// TIA Portal V18 export
VAR_GLOBAL   // PLC tag table "Default tag table"
   ESTOP_Button AT %I0.0 : Bool;   // Emergency button
   JOGNEG_BTN_Z1 AT %I0.2 : Bool;   // Z1 - Jogging Negative -> In order to execute this, real button sholud be pressed
   JOGPOS_BTN_Z1 AT %I0.1 : Bool;   // Z1 - Jogging Positive -> In order to execute this, real button sholud be pressed
   JOGNEG_BTN_Z2 AT %I0.4 : Bool;   // Z2 - Jogging Negative -> In order to execute this, real button sholud be pressed
   JOGPOS_BTN_Z2 AT %I0.3 : Bool;   // Z2 - Jogging Positive -> In order to execute this, real button sholud be pressed
   SENSOR_DOOR AT %I0.5 : Bool;   // Door Sensor Front
   Load_Cell_Ink AT %IW66 : UInt;
   Load_Cell_Waste AT %IW64 : UInt;
   SENSOR_DOOR_2 AT %I0.6 : Bool;   // Door Sensor Front
   UV_Error_Signal AT %I0.7 : Bool;   // Error signal from UV lamp, 0-4 V error, 16-24 V ok;
   SENSOR_DOOR_3 AT %I1.0 : Bool;   // Door Sensor Side
   SENSOR_DOOR_4 AT %I1.1 : Bool;   // Door Sensor Side
   SENSOR_DOOR_5 AT %I1.2 : Bool;   // Door Sensor Fluid Supply
   SENSOR_DOOR_6 AT %I1.3 : Bool;   // Door Sensor Fluid Supply
   TemperatureSensor AT %IW116 : UInt;
   CappingSensor AT %IW118 : UInt;
   AnalogInput3 AT %IW120 : UInt;
   AnalogInput4 AT %IW122 : UInt;
   "Roller Encoder" AT %ID1000 : DWord;
   "STO-B_Output" AT %Q0.0 : Bool;   // Safty Torque Off , for CMMO [Port X3, Pin ..]and CMMP in order to release a break
   Roller_Output AT %Q0.6 : Bool;
   Heater_Output AT %Q1.0 : Bool;   // Heater: ON/OFF_PLC/3.2B; %Q1.0
   LED_1_Output AT %Q0.4 : Bool;
   LED_2_Output AT %Q0.5 : Bool;
   Heater_PWM_pulseduration AT %QW1008 : Int;   // Heater: SETPOINT_PLC/3.2C; %Q0.3
   Capping_Station_PTO AT %Q0.1 : Bool;   //    {ExternalVisible false}
   Capping_Station_DIR AT %Q0.2 : Bool;
   Roller_PWM_pulseduration AT %QW1014 : Int;
   UV_CTRL_ON_OFF AT %Q0.7 : Bool;
   UV_Dimming AT %QW106 : UInt;
   Stacklight01 AT %Q50.0 : Bool;
   Stacklight02 AT %Q50.1 : Bool;
   RollerDirection AT %Q1.1 : Bool;
   Tag_1 AT %IW1000 : Hw_Hsc;
END_VAR
